TEXTLIST FastFadeTime
  0 = 'Disabled'
  4 = 'T100ms'
  8 = 'T200ms'
  12 = 'T300ms'
  16 = 'T400ms'
  20 = 'T500ms'
  24 = 'T600ms'
  27 = 'T700ms'
  255 = 'Unknown'
   = ''
END_TEXTLIST

(* stored: Version 1.1.0.1
   TextList FastFadeTime: Id {794705f7-b70e-4d16-b770-b88f24066f63} *)
